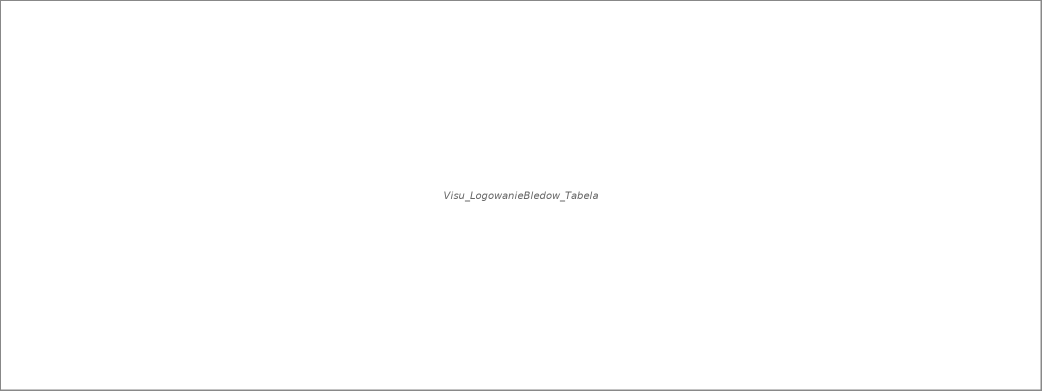
VISUALIZATION Visualization  // 1042x391
    Frame (0,0 1042x391)
        shows Visu_LogowanieBledow_Tabela(stParametry := GVL_LogowanieBledow.fbLoger.stWyswietlanieParametry)
END_VISUALIZATION

(* stored: Version 1.1.0.1, ProductVersion 3.1.4024.11
   Visu Visualization: Id {bb710ff2-8181-4780-bac4-740e17d0ad7e} *)
